TYPE ST_AxisLimit :
STRUCT
	//========================
    // 运动参数允许范围
    // 用于限制上位机输入，保护机械结构
    //========================
    fMinVelocity         : LREAL;//最小速度
    fMaxVelocity         : LREAL;//最大速度

    fMinAcceleration     : LREAL;//最小加速度
    fMaxAcceleration     : LREAL;//最大加速度

    fMinDeceleration     : LREAL;//最小减速度
    fMaxDeceleration     : LREAL;//最大减速度

    //========================
    // 位置限制
    //========================
    fSoftwareLimitPos    : LREAL;//正向软限位
    fSoftwareLimitNeg    : LREAL;//负向软限位
	bSoftLimitEnable 	 : BOOL;// 是否启用PLC侧软限位检查
	fSoftLimitMargin 	 : LREAL;// 点动提前停止的缓冲距离，单位与轴位置单位相同
	bRequireHomed : BOOL;		 // 是否要求轴完成回零
    //========================
    // 力矩限制
    //========================
    fTorqueLimitPos      : LREAL;//最大力矩
    fTorqueLimitNeg      : LREAL;//最小力矩
	
	//========================
    // 跟随误差
    //========================
	fFollowingErrorWarning : LREAL; // 跟随误差警告值
	fFollowingErrorFault   : LREAL; // 跟随误差故障值
	tFollowingErrorDelay   : TIME;  // 超限确认时间
	
	
END_STRUCT
END_TYPE

(* stored: Version 1.1.0.1, ProductVersion 3.1.4026.18
   DUT ST_AxisLimit: Id {0500cab9-42d0-4db2-8fc7-ee74ab6d7f0b} *)
